// TIA Portal V19 export
FUNCTION_BLOCK "F_Estop_FB"   // FB174, F_LAD
// stored: Access Published
   VAR
      ESTOP_CC : ESTOP1;
      ESTOP_A01_FRONT : ESTOP1;
      ESTOP_A01_REAR : ESTOP1;
      ESTOP_A02_FRONT : ESTOP1;
      ESTOP_A02_REAR : ESTOP1;
      ESTOP_A03_FRONT_1 : ESTOP1;
      ESTOP_A03_REAR_1 : ESTOP1;
      ESTOP_A03_FRONT_2 : ESTOP1;
      ESTOP_A03_REAR_2 : ESTOP1;
      ESTOP_A03_FRONT_3 : ESTOP1;
      ESTOP_A03_REAR_3 : ESTOP1;
      EStop : Bool;
      EStop_Delay : Bool;
      F_SafetyValve_Air_Gen : "FDevice_Valve_FB";
   END_VAR
   VAR_TEMP
      Fdbk : Bool;
   END_VAR
   VAR CONSTANT
      TIME_DELAY : Time := T#2s;
   END_VAR
BEGIN

REGION Network 1: ESTOP CC / Leggii
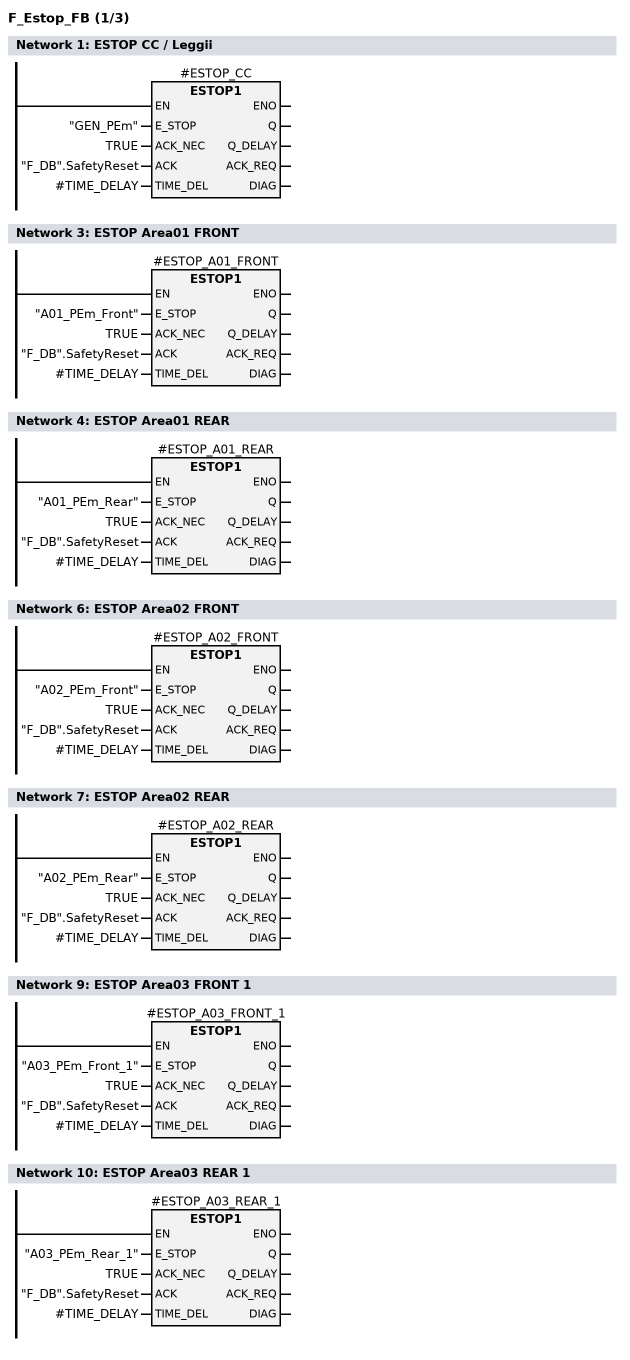
   RUNG wire#powerrail
      #ESTOP_CC.ESTOP1(E_STOP := "GEN_PEm", ACK_NEC := TRUE, ACK := "F_DB".SafetyReset, TIME_DEL := #TIME_DELAY, Q =>, Q_DELAY =>, ACK_REQ =>, DIAG =>)
   END_RUNG
   // the same network as SCL:
   #ESTOP_CC(E_STOP := "GEN_PEm", ACK_NEC := TRUE, ACK := "F_DB".SafetyReset, TIME_DEL := #TIME_DELAY);   // ESTOP1
END_REGION

REGION Network 2: >
END_REGION

REGION Network 3: ESTOP Area01 FRONT
   RUNG wire#powerrail
      #ESTOP_A01_FRONT.ESTOP1(E_STOP := "A01_PEm_Front", ACK_NEC := TRUE, ACK := "F_DB".SafetyReset, TIME_DEL := #TIME_DELAY, Q =>, Q_DELAY =>, ACK_REQ =>, DIAG =>)
   END_RUNG
   // the same network as SCL:
   #ESTOP_A01_FRONT(E_STOP := "A01_PEm_Front",   // ESTOP1
                    ACK_NEC := TRUE,
                    ACK := "F_DB".SafetyReset,
                    TIME_DEL := #TIME_DELAY);
END_REGION

REGION Network 4: ESTOP Area01 REAR
   RUNG wire#powerrail
      #ESTOP_A01_REAR.ESTOP1(E_STOP := "A01_PEm_Rear", ACK_NEC := TRUE, ACK := "F_DB".SafetyReset, TIME_DEL := #TIME_DELAY, Q =>, Q_DELAY =>, ACK_REQ =>, DIAG =>)
   END_RUNG
   // the same network as SCL:
   #ESTOP_A01_REAR(E_STOP := "A01_PEm_Rear",   // ESTOP1
                   ACK_NEC := TRUE,
                   ACK := "F_DB".SafetyReset,
                   TIME_DEL := #TIME_DELAY);
END_REGION

REGION Network 5: >
END_REGION

REGION Network 6: ESTOP Area02 FRONT
   RUNG wire#powerrail
      #ESTOP_A02_FRONT.ESTOP1(E_STOP := "A02_PEm_Front", ACK_NEC := TRUE, ACK := "F_DB".SafetyReset, TIME_DEL := #TIME_DELAY, Q =>, Q_DELAY =>, ACK_REQ =>, DIAG =>)
   END_RUNG
   // the same network as SCL:
   #ESTOP_A02_FRONT(E_STOP := "A02_PEm_Front",   // ESTOP1
                    ACK_NEC := TRUE,
                    ACK := "F_DB".SafetyReset,
                    TIME_DEL := #TIME_DELAY);
END_REGION

REGION Network 7: ESTOP Area02 REAR
   RUNG wire#powerrail
      #ESTOP_A02_REAR.ESTOP1(E_STOP := "A02_PEm_Rear", ACK_NEC := TRUE, ACK := "F_DB".SafetyReset, TIME_DEL := #TIME_DELAY, Q =>, Q_DELAY =>, ACK_REQ =>, DIAG =>)
   END_RUNG
   // the same network as SCL:
   #ESTOP_A02_REAR(E_STOP := "A02_PEm_Rear",   // ESTOP1
                   ACK_NEC := TRUE,
                   ACK := "F_DB".SafetyReset,
                   TIME_DEL := #TIME_DELAY);
END_REGION

REGION Network 8: >
END_REGION

REGION Network 9: ESTOP Area03 FRONT 1
   RUNG wire#powerrail
      #ESTOP_A03_FRONT_1.ESTOP1(E_STOP := "A03_PEm_Front_1", ACK_NEC := TRUE, ACK := "F_DB".SafetyReset, TIME_DEL := #TIME_DELAY, Q =>, Q_DELAY =>, ACK_REQ =>, DIAG =>)
   END_RUNG
   // the same network as SCL:
   #ESTOP_A03_FRONT_1(E_STOP := "A03_PEm_Front_1",   // ESTOP1
                      ACK_NEC := TRUE,
                      ACK := "F_DB".SafetyReset,
                      TIME_DEL := #TIME_DELAY);
END_REGION

REGION Network 10: ESTOP Area03 REAR 1
   RUNG wire#powerrail
      #ESTOP_A03_REAR_1.ESTOP1(E_STOP := "A03_PEm_Rear_1", ACK_NEC := TRUE, ACK := "F_DB".SafetyReset, TIME_DEL := #TIME_DELAY, Q =>, Q_DELAY =>, ACK_REQ =>, DIAG =>)
   END_RUNG
   // the same network as SCL:
   #ESTOP_A03_REAR_1(E_STOP := "A03_PEm_Rear_1",   // ESTOP1
                     ACK_NEC := TRUE,
                     ACK := "F_DB".SafetyReset,
                     TIME_DEL := #TIME_DELAY);
END_REGION

REGION Network 11: ESTOP Area03 FRONT 2
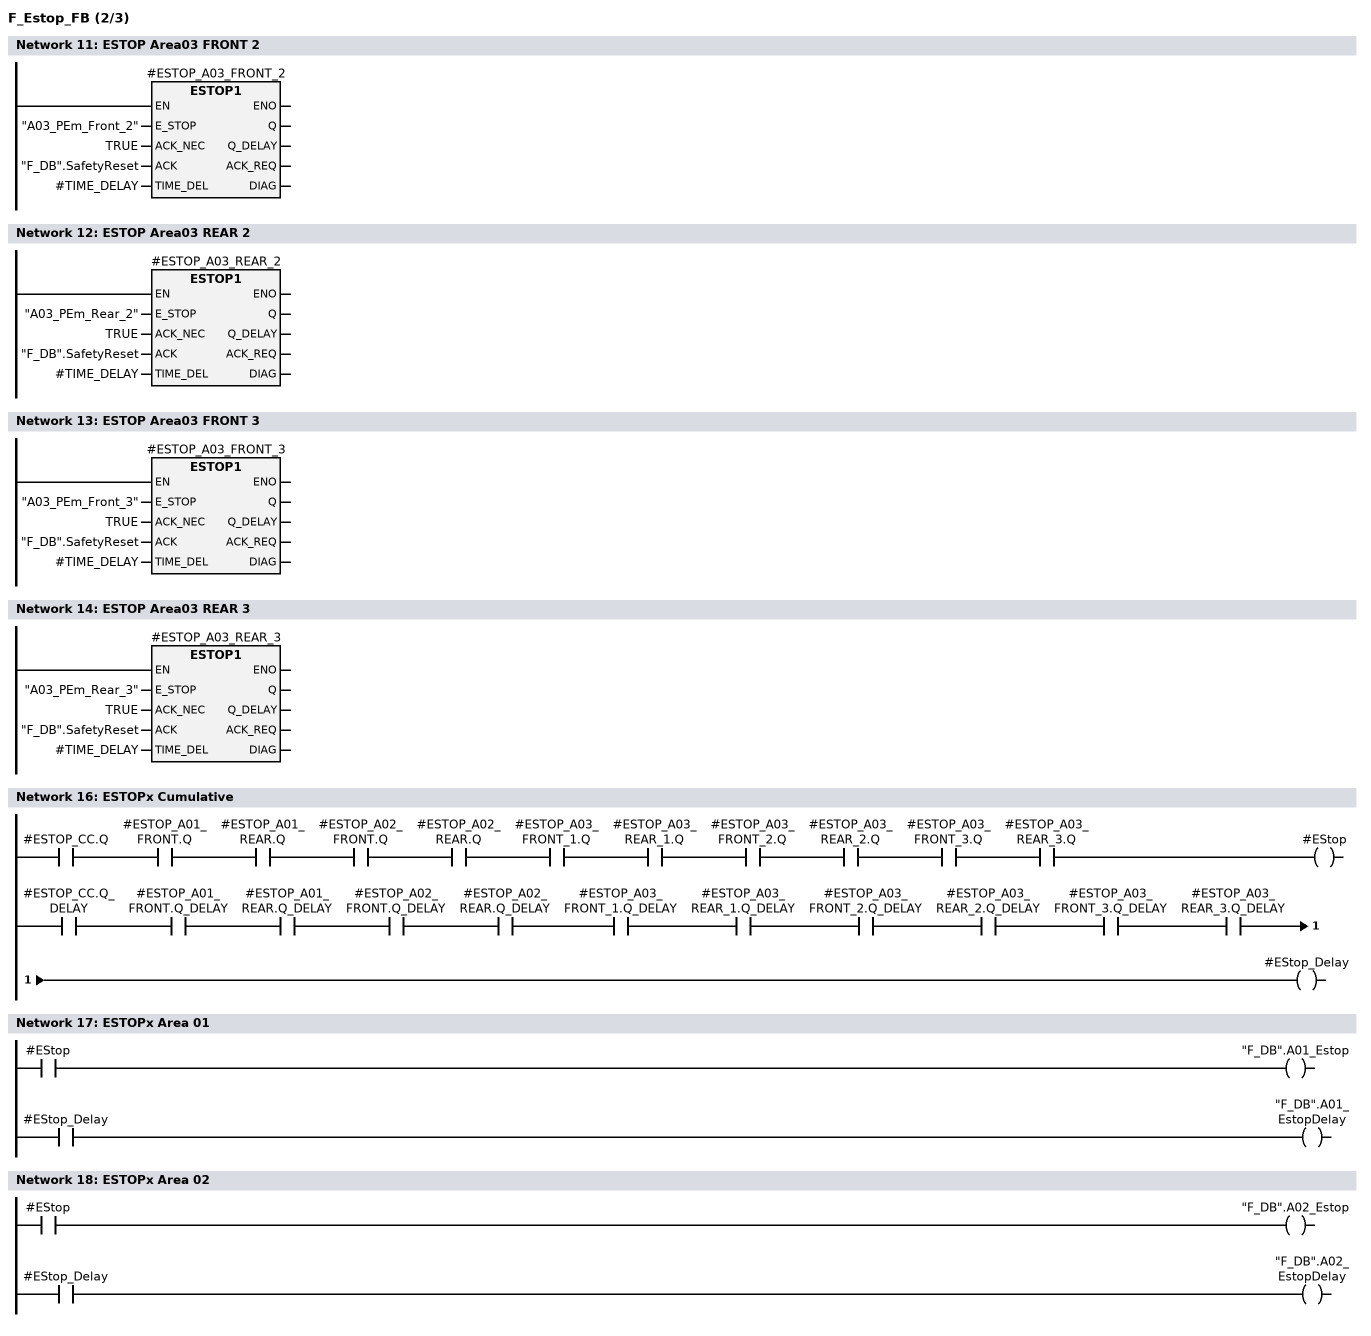
   RUNG wire#powerrail
      #ESTOP_A03_FRONT_2.ESTOP1(E_STOP := "A03_PEm_Front_2", ACK_NEC := TRUE, ACK := "F_DB".SafetyReset, TIME_DEL := #TIME_DELAY, Q =>, Q_DELAY =>, ACK_REQ =>, DIAG =>)
   END_RUNG
   // the same network as SCL:
   #ESTOP_A03_FRONT_2(E_STOP := "A03_PEm_Front_2",   // ESTOP1
                      ACK_NEC := TRUE,
                      ACK := "F_DB".SafetyReset,
                      TIME_DEL := #TIME_DELAY);
END_REGION

REGION Network 12: ESTOP Area03 REAR 2
   RUNG wire#powerrail
      #ESTOP_A03_REAR_2.ESTOP1(E_STOP := "A03_PEm_Rear_2", ACK_NEC := TRUE, ACK := "F_DB".SafetyReset, TIME_DEL := #TIME_DELAY, Q =>, Q_DELAY =>, ACK_REQ =>, DIAG =>)
   END_RUNG
   // the same network as SCL:
   #ESTOP_A03_REAR_2(E_STOP := "A03_PEm_Rear_2",   // ESTOP1
                     ACK_NEC := TRUE,
                     ACK := "F_DB".SafetyReset,
                     TIME_DEL := #TIME_DELAY);
END_REGION

REGION Network 13: ESTOP Area03 FRONT 3
   RUNG wire#powerrail
      #ESTOP_A03_FRONT_3.ESTOP1(E_STOP := "A03_PEm_Front_3", ACK_NEC := TRUE, ACK := "F_DB".SafetyReset, TIME_DEL := #TIME_DELAY, Q =>, Q_DELAY =>, ACK_REQ =>, DIAG =>)
   END_RUNG
   // the same network as SCL:
   #ESTOP_A03_FRONT_3(E_STOP := "A03_PEm_Front_3",   // ESTOP1
                      ACK_NEC := TRUE,
                      ACK := "F_DB".SafetyReset,
                      TIME_DEL := #TIME_DELAY);
END_REGION

REGION Network 14: ESTOP Area03 REAR 3
   RUNG wire#powerrail
      #ESTOP_A03_REAR_3.ESTOP1(E_STOP := "A03_PEm_Rear_3", ACK_NEC := TRUE, ACK := "F_DB".SafetyReset, TIME_DEL := #TIME_DELAY, Q =>, Q_DELAY =>, ACK_REQ =>, DIAG =>)
   END_RUNG
   // the same network as SCL:
   #ESTOP_A03_REAR_3(E_STOP := "A03_PEm_Rear_3",   // ESTOP1
                     ACK_NEC := TRUE,
                     ACK := "F_DB".SafetyReset,
                     TIME_DEL := #TIME_DELAY);
END_REGION

REGION Network 15: >
END_REGION

REGION Network 16: ESTOPx Cumulative
   RUNG wire#powerrail
      Contact( #ESTOP_CC.Q )
      Contact( #ESTOP_A01_FRONT.Q )
      Contact( #ESTOP_A01_REAR.Q )
      Contact( #ESTOP_A02_FRONT.Q )
      Contact( #ESTOP_A02_REAR.Q )
      Contact( #ESTOP_A03_FRONT_1.Q )
      Contact( #ESTOP_A03_REAR_1.Q )
      Contact( #ESTOP_A03_FRONT_2.Q )
      Contact( #ESTOP_A03_REAR_2.Q )
      Contact( #ESTOP_A03_FRONT_3.Q )
      Contact( #ESTOP_A03_REAR_3.Q )
      Coil( #EStop )
   END_RUNG
   RUNG wire#powerrail
      Contact( #ESTOP_CC.Q_DELAY )
      Contact( #ESTOP_A01_FRONT.Q_DELAY )
      Contact( #ESTOP_A01_REAR.Q_DELAY )
      Contact( #ESTOP_A02_FRONT.Q_DELAY )
      Contact( #ESTOP_A02_REAR.Q_DELAY )
      Contact( #ESTOP_A03_FRONT_1.Q_DELAY )
      Contact( #ESTOP_A03_REAR_1.Q_DELAY )
      Contact( #ESTOP_A03_FRONT_2.Q_DELAY )
      Contact( #ESTOP_A03_REAR_2.Q_DELAY )
      Contact( #ESTOP_A03_FRONT_3.Q_DELAY )
      Contact( #ESTOP_A03_REAR_3.Q_DELAY )
      Coil( #EStop_Delay )
   END_RUNG
   // the same network as SCL:
   #EStop := #ESTOP_CC.Q AND #ESTOP_A01_FRONT.Q AND #ESTOP_A01_REAR.Q AND #ESTOP_A02_FRONT.Q AND #ESTOP_A02_REAR.Q AND #ESTOP_A03_FRONT_1.Q AND #ESTOP_A03_REAR_1.Q AND #ESTOP_A03_FRONT_2.Q AND #ESTOP_A03_REAR_2.Q AND #ESTOP_A03_FRONT_3.Q AND #ESTOP_A03_REAR_3.Q;
   #EStop_Delay := #ESTOP_CC.Q_DELAY AND #ESTOP_A01_FRONT.Q_DELAY AND #ESTOP_A01_REAR.Q_DELAY AND #ESTOP_A02_FRONT.Q_DELAY AND #ESTOP_A02_REAR.Q_DELAY AND #ESTOP_A03_FRONT_1.Q_DELAY AND #ESTOP_A03_REAR_1.Q_DELAY AND #ESTOP_A03_FRONT_2.Q_DELAY AND #ESTOP_A03_REAR_2.Q_DELAY AND #ESTOP_A03_FRONT_3.Q_DELAY AND #ESTOP_A03_REAR_3.Q_DELAY;
END_REGION

REGION Network 17: ESTOPx Area 01
   RUNG wire#powerrail
      Contact( #EStop )
      Coil( "F_DB".A01_Estop )
   END_RUNG
   RUNG wire#powerrail
      Contact( #EStop_Delay )
      Coil( "F_DB".A01_EstopDelay )
   END_RUNG
   // the same network as SCL:
   "F_DB".A01_Estop := #EStop;
   "F_DB".A01_EstopDelay := #EStop_Delay;
END_REGION

REGION Network 18: ESTOPx Area 02
   RUNG wire#powerrail
      Contact( #EStop )
      Coil( "F_DB".A02_Estop )
   END_RUNG
   RUNG wire#powerrail
      Contact( #EStop_Delay )
      Coil( "F_DB".A02_EstopDelay )
   END_RUNG
   // the same network as SCL:
   "F_DB".A02_Estop := #EStop;
   "F_DB".A02_EstopDelay := #EStop_Delay;
END_REGION

REGION Network 19: ESTOPx Cumulative Area 03
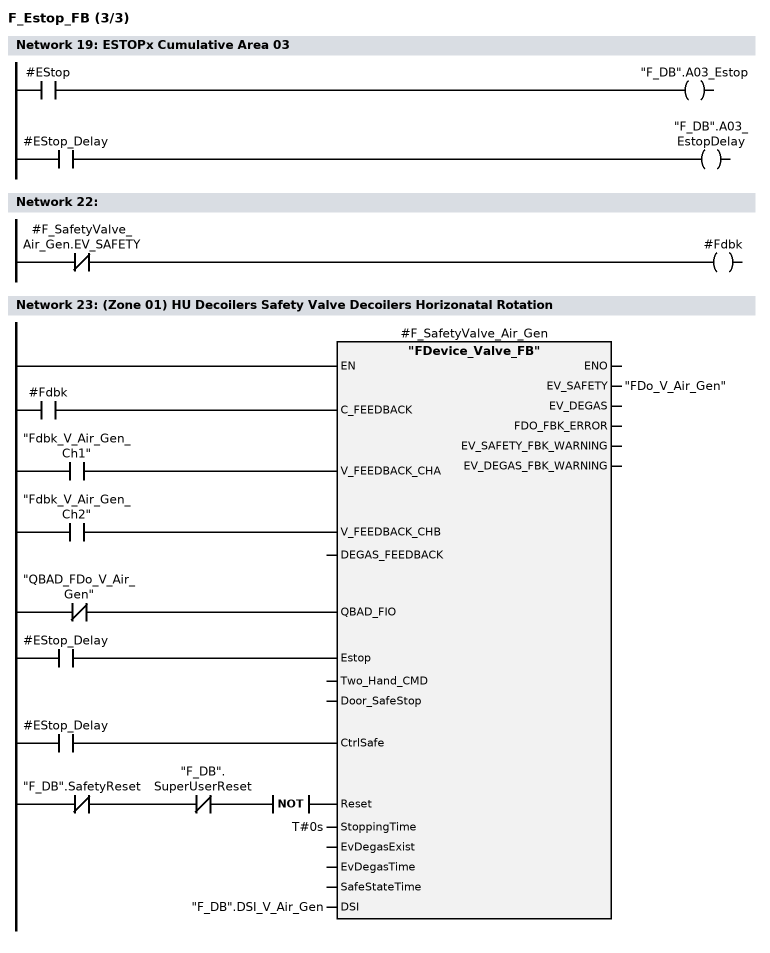
   RUNG wire#powerrail
      Contact( #EStop )
      Coil( "F_DB".A03_Estop )
   END_RUNG
   RUNG wire#powerrail
      Contact( #EStop_Delay )
      Coil( "F_DB".A03_EstopDelay )
   END_RUNG
   // the same network as SCL:
   "F_DB".A03_Estop := #EStop;
   "F_DB".A03_EstopDelay := #EStop_Delay;
END_REGION

REGION Network 20: >
END_REGION

REGION Network 21: < < < < < < < < < < DEVICES SAFETY VALVES > > > > > > > > > >
END_REGION

REGION Network 22
   RUNG wire#powerrail
      I_Contact( #F_SafetyValve_Air_Gen.EV_SAFETY )
      Coil( #Fdbk )
   END_RUNG
   // the same network as SCL:
   #Fdbk := NOT #F_SafetyValve_Air_Gen.EV_SAFETY;
END_REGION

REGION Network 23: (Zone 01) HU Decoilers Safety Valve Decoilers Horizonatal Rotation
   RUNG wire#powerrail
      #F_SafetyValve_Air_Gen(C_FEEDBACK := wire#w1, V_FEEDBACK_CHA := wire#w2, V_FEEDBACK_CHB := wire#w3, QBAD_FIO := wire#w4, Estop := wire#w5, CtrlSafe := wire#w6, Reset := wire#w7, DEGAS_FEEDBACK :=, Two_Hand_CMD :=, Door_SafeStop :=, StoppingTime := T#0s, EvDegasExist :=, EvDegasTime :=, SafeStateTime :=, DSI := "F_DB".DSI_V_Air_Gen, EV_SAFETY => "FDo_V_Air_Gen", EV_DEGAS =>, FDO_FBK_ERROR =>, EV_SAFETY_FBK_WARNING =>, EV_DEGAS_FBK_WARNING =>)
   END_RUNG
   RUNG wire#powerrail
      Contact( #Fdbk )
   END_RUNG wire#w1
   RUNG wire#powerrail
      Contact( "Fdbk_V_Air_Gen_Ch1" )
   END_RUNG wire#w2
   RUNG wire#powerrail
      Contact( "Fdbk_V_Air_Gen_Ch2" )
   END_RUNG wire#w3
   RUNG wire#powerrail
      I_Contact( "QBAD_FDo_V_Air_Gen" )
   END_RUNG wire#w4
   RUNG wire#powerrail
      Contact( #EStop_Delay )
   END_RUNG wire#w5
   RUNG wire#powerrail
      Contact( #EStop_Delay )
   END_RUNG wire#w6
   RUNG wire#powerrail
      I_Contact( "F_DB".SafetyReset )
      I_Contact( "F_DB".SuperUserReset )
      Not()
   END_RUNG wire#w7
   // the same network as SCL:
   #F_SafetyValve_Air_Gen(C_FEEDBACK := #Fdbk,   // "FDevice_Valve_FB"
                          V_FEEDBACK_CHA := "Fdbk_V_Air_Gen_Ch1",
                          V_FEEDBACK_CHB := "Fdbk_V_Air_Gen_Ch2",
                          QBAD_FIO := NOT "QBAD_FDo_V_Air_Gen",
                          Estop := #EStop_Delay,
                          CtrlSafe := #EStop_Delay,
                          Reset := NOT (NOT "F_DB".SafetyReset AND NOT "F_DB".SuperUserReset),
                          StoppingTime := T#0s,
                          DSI := "F_DB".DSI_V_Air_Gen,
                          EV_SAFETY => "FDo_V_Air_Gen");
END_REGION
END_FUNCTION_BLOCK
